(* Logix 5000 project; controller Battleship Emulate 5570 rev 32.11; software revision 32.00 *)

TASK MainTask (continuous, watchdog 500 ms) : MainProgram, Player_2, Player_1

MODULES
   Local : Emulate 5570 (ICP 2, rev 32.11)
END_MODULES

TYPE Bottom_scrn_mod :
STRUCT
   Row0 : Tile[10];
END_STRUCT
END_TYPE

TYPE HMI_ScreenNames :
STRUCT
   LoadingScreen : STRING;
   BattleScreen : STRING;
END_STRUCT
END_TYPE

TYPE PlayerData :
STRUCT
   Ship : Ship[5];
   HMI : PlayerHMI;
   Name : STRING;
   ShipSelectedFromFleet : SINT;
   sideShipSelected_ID : SINT;
   anySideShipSelected : BOOL;
END_STRUCT
END_TYPE

TYPE PlayerHMI :
STRUCT
   Load_Or_Battle : STRING;   // The name of the screen that will load after player presses the Ready button
   ResetBoard : BOOL;
   RetrieveShip : BOOL;
   ShipPiece_Orientation : BOOL;
   Ready : BOOL;   // Player Ready Signal from HMI
   EnableStart : BOOL;   // Enable Start button on HMI
END_STRUCT
END_TYPE

TYPE Ship :
STRUCT
   position : INT[2];   // X-Y Ship Coordinates
   pivot : INT[2];   // X-Y Pivot Coordinates
   shipLength : SINT;   // 5 = Carrier 4 = Battleship 3 = Cruiser 2 = Destroyer
   isHit : BOOL;
   isSunked : BOOL;
   isSelected : BOOL;
   makeSidePieceInvisible : BOOL;
END_STRUCT
END_TYPE

TYPE Tile :
STRUCT
   IND : SINT;   // 0 = No ship 1 = Has ship 2 = Has ship and selected
   ShipID : SINT;
   hasShip : BOOL;
   squareSelected : BOOL;
END_STRUCT
END_TYPE

TYPE top_scrn :
STRUCT
   notSelected : BOOL;
   selected : BOOL;
   hit : BOOL;
END_STRUCT
END_TYPE

TYPE XYcoordinates :
STRUCT
   row : SINT;
   column : SINT;
END_STRUCT
END_TYPE

ADD_ON_INSTRUCTION CommandShip   (* revision 1.0 *)
VAR_IN_OUT
   Player_Ship : Ship[5]; {required}
   Player_tacticalScreen : Tile[10,10]; {required}
END_VAR
VAR_INPUT
   verticalOrientation : BOOL; {required}
   NumberOfShips : DINT; {access Read Only, required}
END_VAR
VAR_IN_OUT
   shipSelected : SINT; {required}
END_VAR
VAR
   selectedSquare : XYcoordinates; {access None}
   x : DINT; {access None}
   row : DINT; {access None}
   column : DINT; {access None}
END_VAR

ROUTINE Logic   (* structured text *)
   // Initialize variables
   //shipSelected := -1;
   selectedSquare.row := -1;
   selectedSquare.column := -1;
   /*
   
   // Look for any side ship that was selected from the side pieces
   // shipSelected = the ship the was selected from the side pieces
   for x := 0 to NumberOfShips-1 by 1  do
   	//anySelected := 0;
   	if Player_Ship[x].isSelected then
   		shipSelected := x;
   		selectedSquare.row := -1;
   		selectedSquare.column := -1;
   	else
   		shipSelected := -1;
   		selectedSquare.row := -1;
   		selectedSquare.column := -1;
   	end_if;
   	/*
   	anySelected := ThisPlayer.Ship[x].isSelected OR anySelected;
   	if not anySelected then
   		shipSelected := -1;
   	end_if;
   
   
   end_for;
   
   */
   
   
   
   // If a ship piece was selected, enable search to look for the square that gets selected on the tactical screen
   // Store the XY coordinates of the selected square in selectedSquare.row and selectedSquare.column
   if shipSelected >= 0 then
   	for row := 0 to 9 by 1 do
   		for column := 0 to 9 by 1 do
   			if Player_tacticalScreen[row,column].squareSelected then
   				selectedSquare.row := row;
   				selectedSquare.column := column;
   				Player_tacticalScreen[row,column].squareSelected := 0;
   			end_if;
   		end_for;
   	end_for;
   end_if;
   
   
   /*
   // If a ship piece and a square were selected,
   // set the adjacent squares "hasShip" to 1 horizontally starting with the selected ship and moving to the right for as many squares as the ship's length
   if selectedSquare.row <> -1 AND selectedSquare.column <> -1 then
   
   	if verticalOrientation then		// Place ship in vertical orientation
   		for column := selectedSquare.column to selectedSquare.column + Player_Ship[x].shipLength -1 by 1 do
   			Player_tacticalScreen[selectedSquare.row,column].hasShip := 1;
   			Player_tacticalScreen[selectedSquare.row,column].hasShipType := shipSelected;
   			Player_tacticalScreen[selectedSquare.row,column].IND := 1;
   			Player_Ship[shipSelected].isSelected := 0;
   		end_for;
   
   
   	else	// Place ship in horizontal orientation
   		for row:= selectedSquare.row to selectedSquare.row + Player_Ship[x].shipLength -1 by 1 do
   			Player_tacticalScreen[row,selectedSquare.column].hasShip := 1;
   			Player_tacticalScreen[row,selectedSquare.column].hasShipType := shipSelected;
   			Player_tacticalScreen[row,selectedSquare.column].IND := 1;
   			Player_Ship[shipSelected].isSelected := 0;
   		end_for;
   	end_if;
   end_if;
   
   
   /*
   TODO
   
   add vertical/horizontal button and adjust how you lay the ship accordingly
   
   add retrieve button
   
   count down the ship pieces. disable piece once count reaches zero
   */
END_ROUTINE
END_ADD_ON_INSTRUCTION

ADD_ON_INSTRUCTION heartBeat   (* revision 1.0 *)
VAR_INPUT
   onTime : DINT; {required}
   offTime : DINT; {required}
END_VAR
VAR_OUTPUT
   Beat : BOOL; {access None, visible}
END_VAR
VAR
   T2 : TIMER; {access None}
   T1 : TIMER; {access None}
END_VAR

ROUTINE Logic   (* ladder *)
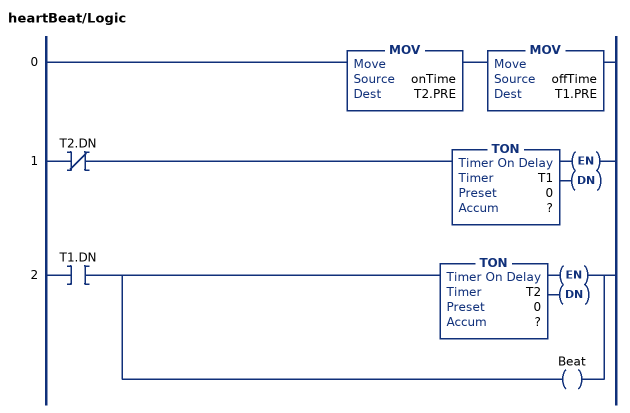
   0: MOV(onTime,T2.PRE)MOV(offTime,T1.PRE);
   1: XIO(T2.DN)TON(T1,?,?);
   2: XIC(T1.DN)[TON(T2,?,?) ,OTE(Beat) ];
END_ROUTINE
END_ADD_ON_INSTRUCTION

ADD_ON_INSTRUCTION ResetTacticalScreen   (* revision 1.0 *)
VAR_IN_OUT
   NULL_TaclticalScreen : Tile; {required}
   P1_tacticalScreen : Tile[10,10]; {required}
END_VAR
VAR
   row : SINT; {access None}
   column : SINT; {access None}
END_VAR

ROUTINE Logic   (* structured text *)
   for row := 0 to 9 by 1 do
   	for column := 0 to 9 by 1 do
   		P1_tacticalScreen[row,column].hasShip := NULL_TaclticalScreen.hasShip;
   		P1_tacticalScreen[row,column].ShipID := NULL_TaclticalScreen.ShipID;
   		P1_tacticalScreen[row,column].IND := NULL_TaclticalScreen.IND;
   		P1_tacticalScreen[row,column].squareSelected := NULL_TaclticalScreen.squareSelected;
   	end_for;
   end_for;
END_ROUTINE
END_ADD_ON_INSTRUCTION

ADD_ON_INSTRUCTION RetrieveShip   (* revision 1.0 *)
VAR_IN_OUT
   Player_tacticalScreen : Tile[10,10]; {required}
END_VAR
VAR_INPUT
   RetrieveShip : BOOL; {required}
END_VAR
VAR
   squareSelected : BOOL; {access None}
   row : DINT; {access None}
   column : DINT; {access None}
   selectedSquare : XYcoordinates; {access None}
   selectedShipType : DINT; {access None}
   readyToRetrieve : BOOL; {access None}
END_VAR

ROUTINE Logic   (* structured text *)
   //Initialize variables
   if not squareSelected then
   	row := -1;
   	column := -1;
   end_if;
   
   
   for row := 0 to 9 by 1 do
   	for column := 0 to 9 by 1 do
   		if Player_tacticalScreen[row,column].squareSelected AND Player_tacticalScreen[row,column].hasShip then
   			selectedSquare.row := row;
   			selectedSquare.column := column;
   			selectedShipType := Player_tacticalScreen[row,column].ShipID;
   			squareSelected := 1;
   			Player_tacticalScreen[row,column].squareSelected := 0;
   		end_if;
   		/*
   		if P1_tacticalScreen[row,column].squareSelected AND P1_tacticalScreen[row,column].IND = 2 then
   			squareSelected := 0;
   			P1_tacticalScreen[row,column].IND := 1;
   		end_if;
   		*/
   	end_for;
   end_for;
   
   
   if squareSelected then
   	for row := 0 to 9 by 1 do
   		for column := 0 to 9 by 1 do
   			if Player_tacticalScreen[row,column].ShipID = selectedShipType then;
   				Player_tacticalScreen[row,column].IND := 2;
   				readyToRetrieve := 1;
   				squareSelected := 0;
   			end_if;
   		end_for;
   	end_for;
   end_if;
   
   if readyToRetrieve AND RetrieveShip then
   	for row := 0 to 9 by 1 do
   		for column := 0 to 9 by 1 do
   			if Player_tacticalScreen[row,column].ShipID = selectedShipType then;
   				Player_tacticalScreen[row,column].hasShip := 0;
   				Player_tacticalScreen[row,column].IND := 0;
   				Player_tacticalScreen[row,column].ShipID := -1;
   				readyToRetrieve := 0;
   				squareSelected := 0;
   			end_if;
   		end_for;
   	end_for;
   end_if;
   
   
   if squareSelected AND Player_tacticalScreen[selectedSquare.row,selectedSquare.column].IND = 2 then
   	for row := 0 to 9 by 1 do
   		for column := 0 to 9 by 1 do
   			if Player_tacticalScreen[row,column].ShipID = selectedShipType then;
   				Player_tacticalScreen[row,column].IND := 1;
   				readyToRetrieve := 0;
   				squareSelected := 0;
   			end_if;
   		end_for;
   	end_for;
   end_if;
   
END_ROUTINE
END_ADD_ON_INSTRUCTION

ADD_ON_INSTRUCTION SideShips   (* revision 1.0 *)
VAR_IN_OUT
   Player_Ship : Ship[5]; {required}
END_VAR
VAR_OUTPUT
   shipSelected : SINT; {required}
END_VAR
VAR
   shipCount : SINT; {access None}
   shipSelected_OSR : FBD_ONESHOT[9]; {access None}
   aShipWasSelected : BOOL[32]; {access None}
END_VAR

ROUTINE Logic   (* structured text *)
   // This code handles the ship pieces tha get selected on the left of the tactical screen
   
   // Look for a one shot rising that comes from pressing on one ship piece. Save which ship piece was selected to shipSelected
   
   
   for shipCount:=0 to 8 by 1 do
   	if not Player_Ship[shipCount].isSelected then
   		shipSelected := -1;
   	end_if;
   
   	shipSelected_OSR[shipCount].InputBit := Player_Ship[shipCount].isSelected;
   	OSRI(shipSelected_OSR[shipCount]);
   	aShipWasSelected[shipCount] := shipSelected_OSR[shipCount].OutputBit;
   
   	if aShipWasSelected[shipCount] then
   		shipSelected := shipCount;
   	end_if;
   end_for;
   
   
   if aShipWasSelected[0] or aShipWasSelected[1] or aShipWasSelected[2] or aShipWasSelected[3] or aShipWasSelected[4] or aShipWasSelected[5] then
   	aShipWasSelected[10] := 1;
   end_if;
   
   if aShipWasSelected[6] or aShipWasSelected[7] or aShipWasSelected[8] or aShipWasSelected[9] then
   	aShipWasSelected[11] := 1;
   end_if;
   
   // If ANY ship was selected then NONE of the other ships can be selected, set isSelected (for the rest of the ships) to zero
   if aShipWasSelected[10] or aShipWasSelected[11] then
   	for shipCount:=0 to 8 by 1 do
   		if shipCount <> shipSelected then
   			Player_Ship[shipCount].isSelected := 0;
   		end_if;
   	end_for;
   end_if;
   
   /*
   TODO
   
   Keep count of how many ship pieces are left
   */
END_ROUTINE
END_ADD_ON_INSTRUCTION

ADD_ON_INSTRUCTION TacticalScreen_TileDetection   (* revision 1.0 *)
VAR_IN_OUT
   TacticalScreen : Tile[10,10]; {required}
   selectedSquare : XYcoordinates; {required}
   SelectedTileShipID : DINT; {required}
END_VAR
VAR
   row : DINT; {access None}
   column : DINT; {access None}
END_VAR

ROUTINE Logic   (* structured text *)
   /*
   -------------------------------------------------------------------------------------------------
   	This FB Scans the Tactical Screen and returns the X-Y coordinates of the tile that was selected
   	It also returns the ShipID of the ship placed in the selected tile
   
   
   -------------------------------------------------------------------------------------------------
   */
   
   
   for row := 0 to 9 by 1 do
   	for column := 0 to 9 by 1 do
   		if TacticalScreen[row,column].squareSelected then
   
   			selectedSquare.row := row;
   			selectedSquare.column := column;
   			SelectedTileShipID := TacticalScreen[row,column].ShipID;
   
   		end_if;
   	end_for;
   end_for;
END_ROUTINE
END_ADD_ON_INSTRUCTION

VAR_GLOBAL   (* controller tags *)
   anySelected : BOOL;
   column : DINT := 10;
   HeartBeat : BOOL;
   NULL_TaclticalScreen : Tile := (ShipID := -1); {access Read Only}
   NumberOfShips : SINT := 5; {constant, access Read Only}
   P1_TacticalScreen : Tile[10,10] := ([0,0].ShipID := -1, [0,1].ShipID := -1, [0,2].ShipID := -1, [0,3].ShipID := -1, [0,4].ShipID := -1, [0,5].ShipID := -1, [0,6].ShipID := -1, [0,7].ShipID := -1, [0,8].ShipID := -1, [0,9].ShipID := -1, [1,0].ShipID := -1, [1,1].ShipID := -1, [1,2].ShipID := -1, [1,3].ShipID := -1, [1,4].ShipID := -1, [1,5].ShipID := -1, [1,6].ShipID := -1, [1,7].ShipID := -1, [1,8].ShipID := -1, [1,9].ShipID := -1, [2,0].ShipID := -1, [2,1].ShipID := -1, [2,2].ShipID := -1, [2,3].ShipID := -1, [2,4].ShipID := -1, [2,5].ShipID := -1, [2,6].ShipID := -1, [2,7].ShipID := -1, [2,8].ShipID := -1, [2,9].ShipID := -1, [3,0].ShipID := -1, [3,1].ShipID := -1, [3,2].ShipID := -1, [3,3].ShipID := -1, [3,4].ShipID := -1, [3,5].ShipID := -1, [3,6].ShipID := -1, [3,7].ShipID := -1, [3,8].ShipID := -1, [3,9].ShipID := -1, [4,0].ShipID := -1, [4,1].ShipID := -1, [4,2].ShipID := -1, [4,3].ShipID := -1, [4,4].ShipID := -1, [4,5].ShipID := -1, [4,6].ShipID := -1, [4,7].ShipID := -1, [4,8].ShipID := -1, [4,9].ShipID := -1, [5,0].ShipID := -1, [5,1].ShipID := -1, [5,2].ShipID := -1, [5,3].ShipID := -1, [5,4].ShipID := -1, [5,5].ShipID := -1, [5,6].ShipID := -1, [5,7].ShipID := -1, [5,8].ShipID := -1, [5,9].ShipID := -1,
        [6,0].ShipID := -1, [6,1].ShipID := -1, [6,2].ShipID := -1, [6,3].ShipID := -1, [6,4].ShipID := -1, [6,5].ShipID := -1, [6,6].ShipID := -1, [6,7].ShipID := -1, [6,8].ShipID := -1, [6,9].ShipID := -1, [7,0].ShipID := -1, [7,1].ShipID := -1, [7,2].ShipID := -1, [7,3].ShipID := -1, [7,4].ShipID := -1, [7,5].ShipID := -1, [7,6].ShipID := -1, [7,7].ShipID := -1, [7,8].ShipID := -1, [7,9].ShipID := -1, [8,0].ShipID := -1, [8,1].ShipID := -1, [8,2].ShipID := -1, [8,3].ShipID := -1, [8,4].ShipID := -1, [8,5].ShipID := -1, [8,6].ShipID := -1, [8,7].ShipID := -1, [8,8].ShipID := -1, [8,9].ShipID := -1, [9,0].ShipID := -1, [9,1].ShipID := -1, [9,2].ShipID := -1, [9,3].ShipID := -1, [9,4].ShipID := -1, [9,5].ShipID := -1, [9,6].ShipID := -1, [9,7].ShipID := -1, [9,8].ShipID := -1, [9,9].ShipID := -1);
   Player1 : PlayerData := (Ship[0].shipLength := 5, Ship[1].shipLength := 4, Ship[2].shipLength := 3, Ship[3].shipLength := 3, Ship[4].shipLength := 2, HMI.Load_Or_Battle := '0_LoadinScreen', HMI.ShipPiece_Orientation := 1, sideShipSelected_ID := -1);
   Player2 : PlayerData := (sideShipSelected_ID := -1);
   row : DINT := 3;
   ScreenNamesData : HMI_ScreenNames := (LoadingScreen := '0_LoadinScreen', BattleScreen := '1_BattleScreen');
   selectedSquare : XYcoordinates := (row := -1, column := -1);
   SelectedTileShipID : SINT;
   Ship_NULL : Ship;
END_VAR

PROGRAM MainProgram   (* main routine MainRoutine *)
VAR
   Heart : heartBeat := (onTime := 500, offTime := 500);
END_VAR

ROUTINE MainRoutine   (* ladder *)
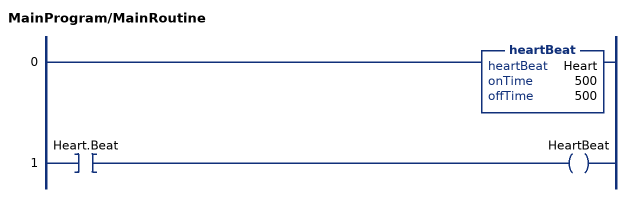
   0: heartBeat(Heart,500,500);
   1: XIC(Heart.Beat)OTE(HeartBeat);
END_ROUTINE

ROUTINE Score   (* function block diagram *)
   SHEET 1
END_ROUTINE
END_PROGRAM

PROGRAM Player_1   (* main routine Main *)
VAR
   AOI_TileDetection : TacticalScreen_TileDetection; {access Read Only}
   cntr : SINT := 5;
   CycleLoadingTime : DINT := 5000;
   DotOff : SINT := 64;
   DotOff_Time : REAL[8] := ([0] := 625.0, [1] := 1250.0, [2] := 1875.0, [3] := 2500.0, [4] := 3125.0, [5] := 3750.0, [6] := 4375.0, [7] := 5000.0);
   LoadingDots : TIMER := (PRE := 5000, ACC := 4009, EN := 1, TT := 1);
        .PRE   // Use this to change how fast the loading dots move
   OtherPlayer : ALIAS FOR Player2;
   pResetBoard_ONS : BOOL; {access Read Only}
   ResetScreen : ResetTacticalScreen; {access Read Only}
   RetrieveShips : RetrieveShip;   // Handles ship retrieving process
   rtrv_column : DINT; {access Read Only}
   rtrv_column2 : DINT; {access Read Only}
   rtrv_row : DINT; {access Read Only}
   rtrv_row2 : DINT; {access Read Only}
   rtv_selectedSquare : XYcoordinates; {access Read Only}
   shipSelected_OSR : FBD_ONESHOT[15];
   shipUnselected_OSR : FBD_ONESHOT[15];
   TacticalScreen_SelectedTile : XYcoordinates; {access Read Only}
   TacticalScreen_SelectedTile_ShipID : DINT; {access Read Only}
   ThisPlayer : ALIAS FOR Player1;
END_VAR

ROUTINE HMI   (* ladder *)
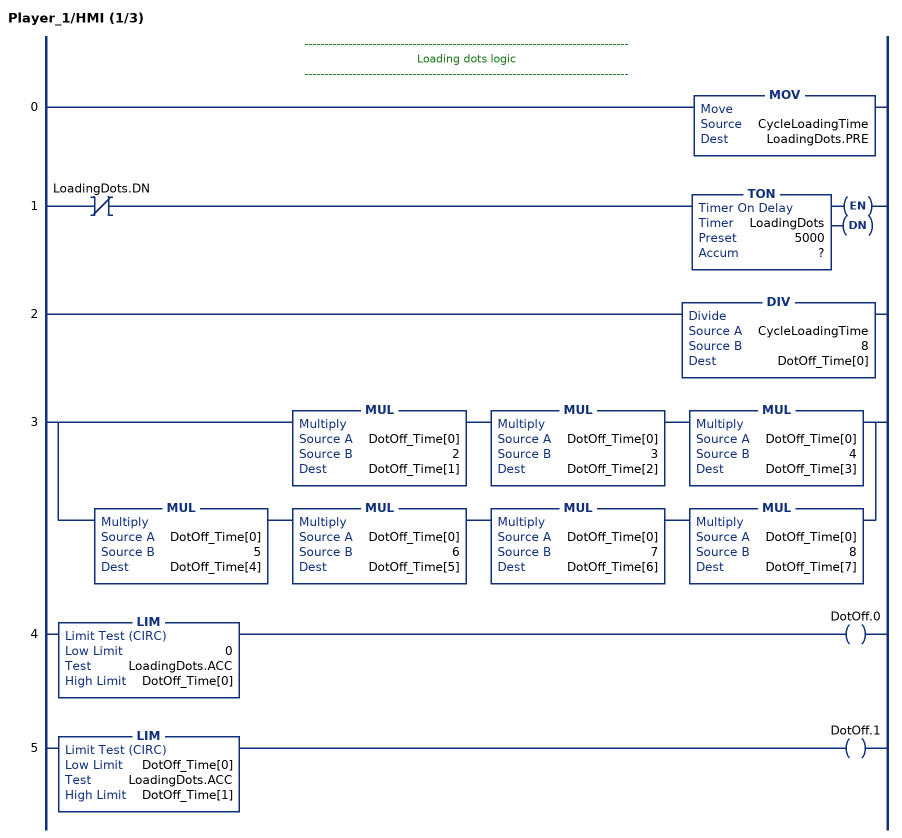
   // ---------------------------------------------------------------------------------
   // Loading dots logic
   // ---------------------------------------------------------------------------------
   0: MOV(CycleLoadingTime,LoadingDots.PRE);
   1: XIO(LoadingDots.DN)TON(LoadingDots,?,?);
   2: DIV(CycleLoadingTime,8,DotOff_Time[0]);
   3: [MUL(DotOff_Time[0],2,DotOff_Time[1]) MUL(DotOff_Time[0],3,DotOff_Time[2]) MUL(DotOff_Time[0],4,DotOff_Time[3]) ,MUL(DotOff_Time[0],5,DotOff_Time[4]) MUL(DotOff_Time[0],6,DotOff_Time[5]) MUL(DotOff_Time[0],7,DotOff_Time[6]) MUL(DotOff_Time[0],8,DotOff_Time[7]) ];
   4: LIM(0,LoadingDots.ACC,DotOff_Time[0])OTE(DotOff.0);
   5: LIM(DotOff_Time[0],LoadingDots.ACC,DotOff_Time[1])OTE(DotOff.1);
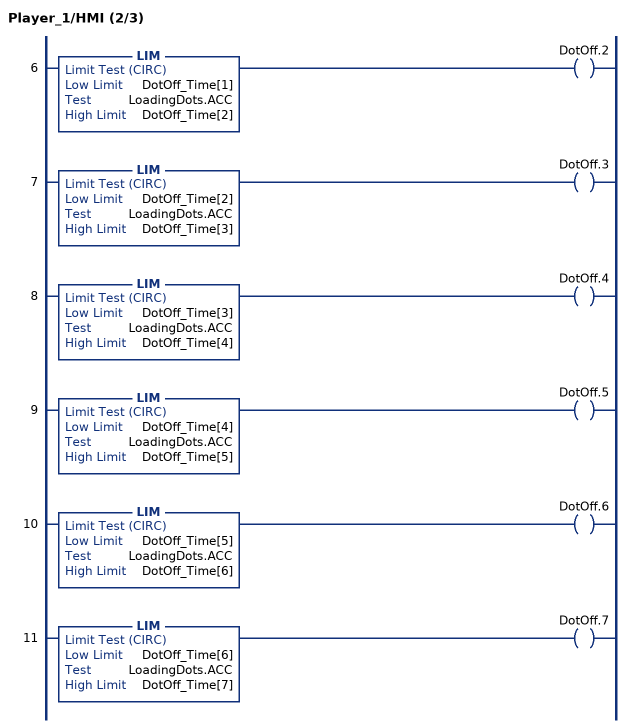
   6: LIM(DotOff_Time[1],LoadingDots.ACC,DotOff_Time[2])OTE(DotOff.2);
   7: LIM(DotOff_Time[2],LoadingDots.ACC,DotOff_Time[3])OTE(DotOff.3);
   8: LIM(DotOff_Time[3],LoadingDots.ACC,DotOff_Time[4])OTE(DotOff.4);
   9: LIM(DotOff_Time[4],LoadingDots.ACC,DotOff_Time[5])OTE(DotOff.5);
   10: LIM(DotOff_Time[5],LoadingDots.ACC,DotOff_Time[6])OTE(DotOff.6);
   11: LIM(DotOff_Time[6],LoadingDots.ACC,DotOff_Time[7])OTE(DotOff.7);
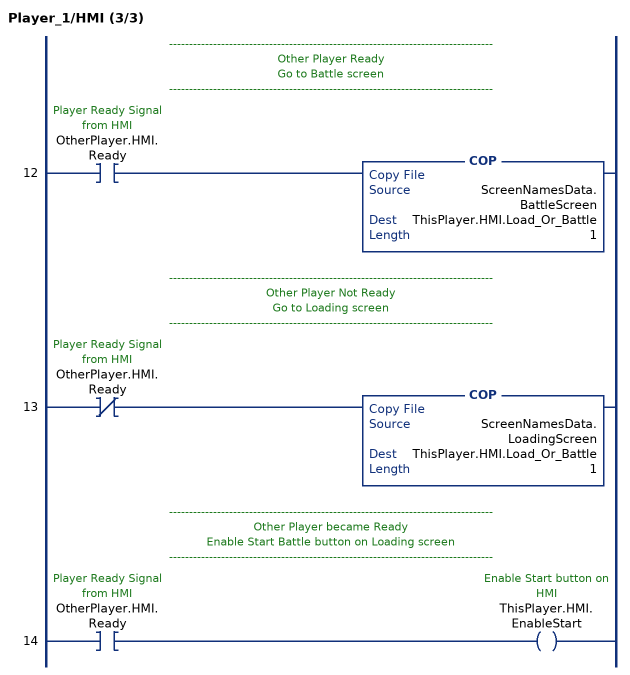
   // ---------------------------------------------------------------------------------
   // Other Player Ready
   // Go to Battle screen
   // ---------------------------------------------------------------------------------
   12: XIC(OtherPlayer.HMI.Ready)COP(ScreenNamesData.BattleScreen,ThisPlayer.HMI.Load_Or_Battle,1);
   // ---------------------------------------------------------------------------------
   // Other Player Not Ready
   // Go to Loading screen
   // ---------------------------------------------------------------------------------
   13: XIO(OtherPlayer.HMI.Ready)COP(ScreenNamesData.LoadingScreen,ThisPlayer.HMI.Load_Or_Battle,1);
   // ---------------------------------------------------------------------------------
   // Other Player became Ready
   // Enable Start Battle button on Loading screen
   // ---------------------------------------------------------------------------------
   14: XIC(OtherPlayer.HMI.Ready)OTE(ThisPlayer.HMI.EnableStart);
END_ROUTINE

ROUTINE Main   (* ladder *)
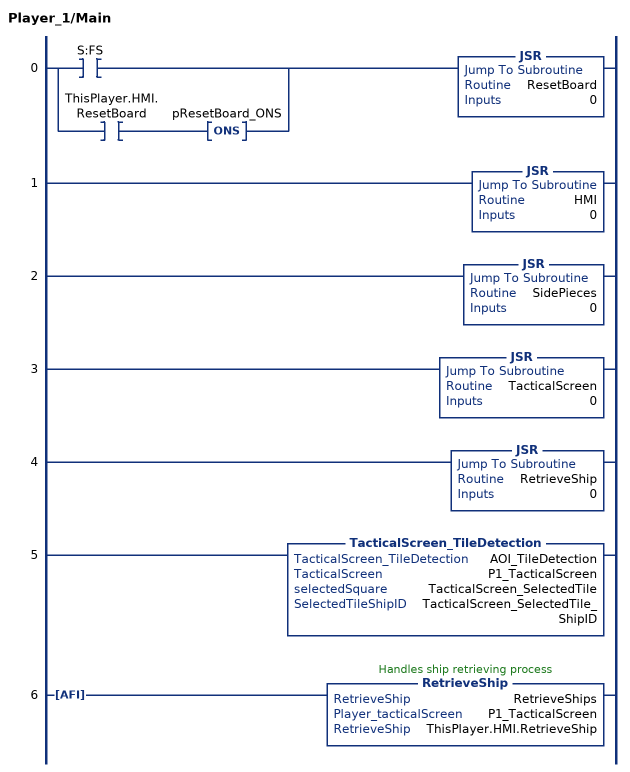
   0: [XIC(S:FS) ,XIC(ThisPlayer.HMI.ResetBoard) ONS(pResetBoard_ONS) ]JSR(ResetBoard,0);
   1: JSR(HMI,0);
   2: JSR(SidePieces,0);
   3: JSR(TacticalScreen,0);
   4: JSR(RetrieveShip,0);
   5: TacticalScreen_TileDetection(AOI_TileDetection,P1_TacticalScreen,TacticalScreen_SelectedTile,TacticalScreen_SelectedTile_ShipID);
   6: AFI()RetrieveShip(RetrieveShips,P1_TacticalScreen,ThisPlayer.HMI.RetrieveShip);
END_ROUTINE

ROUTINE ResetBoard   (* ladder *)
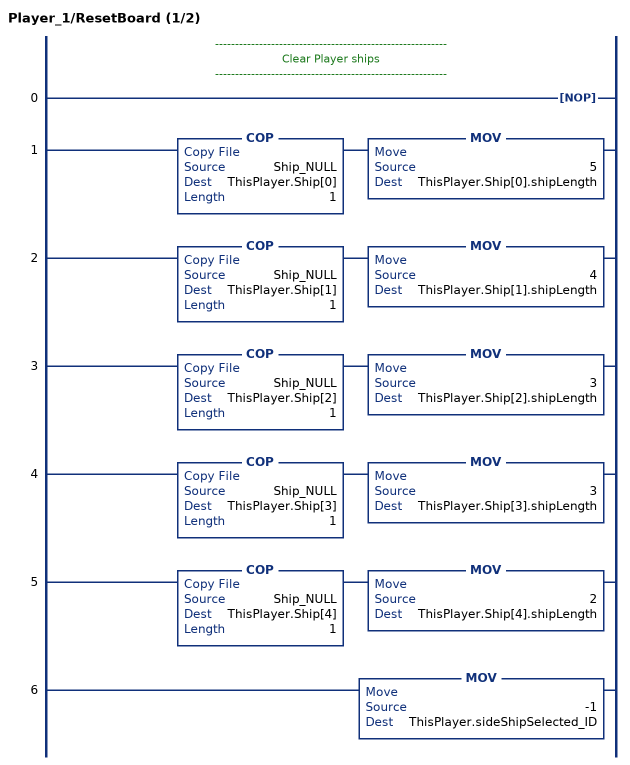
   // ----------------------------------------------------------
   // Clear Player ships
   // ----------------------------------------------------------
   0: NOP();
   1: COP(Ship_NULL,ThisPlayer.Ship[0],1)MOV(5,ThisPlayer.Ship[0].shipLength);
   2: COP(Ship_NULL,ThisPlayer.Ship[1],1)MOV(4,ThisPlayer.Ship[1].shipLength);
   3: COP(Ship_NULL,ThisPlayer.Ship[2],1)MOV(3,ThisPlayer.Ship[2].shipLength);
   4: COP(Ship_NULL,ThisPlayer.Ship[3],1)MOV(3,ThisPlayer.Ship[3].shipLength);
   5: COP(Ship_NULL,ThisPlayer.Ship[4],1)MOV(2,ThisPlayer.Ship[4].shipLength);
   6: MOV(-1,ThisPlayer.sideShipSelected_ID);
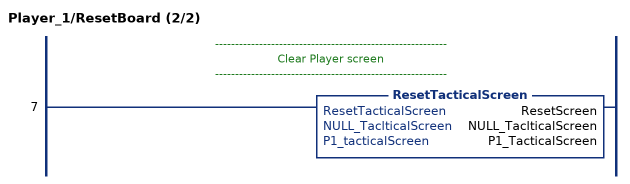
   // ----------------------------------------------------------
   // Clear Player screen
   // ----------------------------------------------------------
   7: ResetTacticalScreen(ResetScreen,NULL_TaclticalScreen,P1_TacticalScreen);
END_ROUTINE

ROUTINE RetrieveShip   (* structured text *)
   //Initialize variables
   /*
   if not anySelected then
   	rtrv_row := -1;
   	rtrv_column := -1;
   end_if;
   */
   
   
   for rtrv_row := 0 to 9 by 1 do
   	for rtrv_column := 0 to 9 by 1 do
   		if P1_TacticalScreen[rtrv_row,rtrv_column].squareSelected AND P1_TacticalScreen[rtrv_row,rtrv_column].hasShip and not anySelected then
   
   			rtv_selectedSquare.row := rtrv_row;
   			rtv_selectedSquare.column := rtrv_column;
   			SelectedTileShipID := P1_TacticalScreen[rtrv_row,rtrv_column].ShipID;
   			anySelected := 1;
   			P1_TacticalScreen[rtrv_row,rtrv_column].squareSelected := 0;
   
   		end_if;
   	end_for;
   end_for;
   
   if anySelected then
   	for rtrv_row := 0 to 9 by 1 do
   		for rtrv_column := 0 to 9 by 1 do
   			if P1_TacticalScreen[rtrv_row,rtrv_column].ShipID = SelectedTileShipID then;
   				P1_TacticalScreen[rtrv_row,rtrv_column].IND := 2;
   
   				if P1_TacticalScreen[rtrv_row,rtrv_column].squareSelected then;
   					for rtrv_row2 := 0 to 9 by 1 do
   						for rtrv_column2 := 0 to 9 by 1 do
   							if P1_TacticalScreen[rtrv_row2,rtrv_column2].ShipID = SelectedTileShipID then;
   
   								P1_TacticalScreen[rtrv_row2,rtrv_column2].IND := 1;
   							end_if;
   						end_for;
   					end_for;
   					P1_TacticalScreen[rtrv_row,rtrv_column].squareSelected := 0;
   					anySelected := 0;
   				end_if;
   
   
   
   				if ThisPlayer.HMI.RetrieveShip then
   					//TileShipID := P1_TacticalScreen[rtrv_row,rtrv_column].hasShipType;
   					ThisPlayer.Ship[SelectedTileShipID].makeSidePieceInvisible := 0;
   					P1_TacticalScreen[rtrv_row,rtrv_column].ShipID := -1;
   					P1_TacticalScreen[rtrv_row,rtrv_column].hasShip := 0;
   					P1_TacticalScreen[rtrv_row,rtrv_column].IND := 0;
   					anySelected := 0;
   
   
   
   				end_if;
   			end_if;
   		end_for;
   	end_for;
   end_if;
END_ROUTINE

ROUTINE SidePieces   (* structured text *)
   /*
   -------------------------------------------------------------------------------------------------------------------------------------------------------------------
   This code handles the ship pieces tha get selected on the left of the tactical screen
   
   When a piece is selected, one of the (10) one shot rising (one for every ship) gets triggered and the ship's ID number gets recorded in ThisPlayer.sideShipSelected_ID
   The counter will match the ship ID number for whichever gets triggered
   
   one of the 10 one shot falling will record if a ship gets unselected, when that happens the ship ID will go to 0
   
   We assing a 0 to every ship that's not selected, since only one can be selected at any given time
   -------------------------------------------------------------------------------------------------------------------------------------------------------------------
   */
   
   for cntr := 0 to NumberOfShips-1 by 1 do								// Scan from ship 0 to the last ship
   
   
   	shipSelected_OSR[cntr].InputBit := ThisPlayer.Ship[cntr].isSelected;
   	OSRI(shipSelected_OSR[cntr]);
   	if shipSelected_OSR[cntr].OutputBit then
   		ThisPlayer.sideShipSelected_ID := cntr;		// Capture the ID of the piece selected
   	end_if;
   
   
   	if cntr <> ThisPlayer.sideShipSelected_ID then
   		ThisPlayer.Ship[cntr].isSelected := 0;			// Set the rest to zero
   	end_if;
   
   
   
   	shipUnselected_OSR[cntr].InputBit := ThisPlayer.Ship[cntr].isSelected;
   	OSFI(shipUnselected_OSR[cntr]);
   
   	if shipUnselected_OSR[cntr].OutputBit and 	ThisPlayer.sideShipSelected_ID = cntr then		// Set ID to zero if a piece that was selected has a OSF
   		ThisPlayer.sideShipSelected_ID := -1;
   	end_if;
   
   
   end_for;
   
   /*
   TODO
   make pieces invisible when put on the board
   */
END_ROUTINE

ROUTINE TacticalScreen   (* structured text *)
   /*
   // Initialize variables
   if not anySelected then
   	shipSelected := -1;
   	selectedSquare.row := -1;
   	selectedSquare.column := -1;
   end_if;
   
   // Look for any side ship that was selected from the side pieces
   // shipSelected = the ship the was selected from the side pieces
   for x := 0 to NumberOfShips-1 by 1  do
   	//anySelected := 0;
   	if ThisPlayer.Ship[x].isSelected then
   		shipSelected := x;
   	end_if;
   	/*
   	anySelected := ThisPlayer.Ship[x].isSelected OR anySelected;
   	if not anySelected then
   		shipSelected := -1;
   	end_if;
   
   
   end_for;
   */
   
   // If a ship piece was selected, enable search to look for the square that gets selected on the tactical screen
   // Store the XY coordinates of the selected square in selectedSquare.row and selectedSquare.column
   if ThisPlayer.sideShipSelected_ID >= 0 then
   	for row := 0 to 9 by 1 do
   		for column := 0 to 9 by 1 do
   			if P1_TacticalScreen[row,column].squareSelected then
   				selectedSquare.row := row;
   				selectedSquare.column := column;
   				P1_TacticalScreen[row,column].squareSelected := 0;
   			end_if;
   		end_for;
   	end_for;
   else
   	selectedSquare.row := -1;
   	selectedSquare.column := -1;
   end_if;
   
   // If a ship piece and a square were selected,
   // set the adjacent squares "hasShip" to 1 horizontally starting with the selected ship and moving to the left for as many squares as the ship's length
   if selectedSquare.row <> -1 AND selectedSquare.column <> -1 then
   
   	if ThisPlayer.HMI.ShipPiece_Orientation then		// Place ship in vertical orientation
   		for row := selectedSquare.row to selectedSquare.row + ThisPlayer.Ship[ThisPlayer.sideShipSelected_ID].shipLength -1 by 1 do
   			P1_TacticalScreen[row,selectedSquare.column].hasShip := 1;
   			P1_TacticalScreen[row,selectedSquare.column].ShipID := ThisPlayer.sideShipSelected_ID;
   			P1_TacticalScreen[row,selectedSquare.column].IND := 1;
   			ThisPlayer.Ship[ThisPlayer.sideShipSelected_ID].isSelected := 0;
   		end_for;
   
   
   	else	// Place ship in horizontal orientation
   		for column := selectedSquare.column to selectedSquare.column + ThisPlayer.Ship[ThisPlayer.sideShipSelected_ID].shipLength -1 by 1 do
   			P1_TacticalScreen[selectedSquare.row,column].hasShip := 1;
   			P1_TacticalScreen[selectedSquare.row,column].ShipID := ThisPlayer.sideShipSelected_ID;
   			P1_TacticalScreen[selectedSquare.row,column].IND := 1;
   			ThisPlayer.Ship[ThisPlayer.sideShipSelected_ID].isSelected := 0;
   		end_for;
   	end_if;
   
   
   	ThisPlayer.Ship[ThisPlayer.sideShipSelected_ID].makeSidePieceInvisible := 1;
   
   end_if;
   
   
   /*
   TODO
   
   add vertical/horizontal button and adjust how you lay the ship accordingly
   
   add retrieve button
   
   count down the ship pieces. disable piece once count reaches zero
   */
END_ROUTINE
END_PROGRAM

PROGRAM Player_2   (* main routine Main *)

ROUTINE Main   (* ladder *)
END_ROUTINE
END_PROGRAM
